// TwinCAT 3 PLC project ASRS_2
// ProgramVersion: 3.1.4024.0
// libraries:
//   Tc2_Standard, * (Beckhoff Automation GmbH)
//   Tc2_System, * (Beckhoff Automation GmbH)
//   Tc3_Module, * (Beckhoff Automation GmbH)
// project tree:
//   DUTs/Enum/ E_ConveyorMode.TcDUT, E_DiverterState.TcDUT (not stored), E_CraneState.TcDUT (not stored), E_AisleMode.TcDUT (not stored), E_SlotStatus.TcDUT (not stored), E_WarehouseState.TcDUT (not stored)
//   DUTs/Structure/ ST_Parcel.TcDUT (not stored), ST_StorageSlot.TcDUT (not stored), ST_Position.TcDUT (not stored), ST_CraneJob.TcDUT (not stored), ST_HMI_Search.TcDUT
//   GVLs/ GVL_IO.TcGVL, GVL_Config.TcGVL (not stored), GVL_Warehouse.TcGVL
//   / PlcTask.TcTTO (not stored)
//   POUs/ Class Diagram.TcCD (not stored), FB_WareHouseController.TcPOU, MAIN.TcPOU
//   POUs/ITFs/ I_Conveyor.TcIO, I_Diverter.TcIO (not stored), I_Crane.TcIO (not stored)
//   POUs/Entity/ FB_Conveyor.TcPOU, FB_BiDirectionConveyor.TcPOU (not stored), FB_RAT.TcPOU, FB_Crane.TcPOU (not stored)
//   POUs/Controller/ FB_InFeedController.TcPOU, FB_LoopController.TcPOU, FB_AisleController.TcPOU (not stored), FB_CraneController.TcPOU (not stored), FB_OutFeedController.TcPOU
// (motion and I/O tree: see PLC project asrs_test)
// real-time tasks:
//   TASK PlcTask: cycle T#10ms, priority 20, ADS port 350
//   TASK PlcTask1: cycle T#10ms, priority 21, ADS port 351

// ---- DUTs/Enum/E_ConveyorMode.TcDUT
{attribute 'qualified_only'}
{attribute 'strict'}
TYPE E_ConveyorMode :
(
    IDLE              := 0,
    RUNNING_FORWARD   := 10,
    RUNNING_BACKWARD  := 20,
    FAULT             := 99
);
END_TYPE

// ---- DUTs/Structure/ST_HMI_Search.TcDUT
TYPE ST_HMI_Search :
STRUCT
    (* Input from Operator *)
    sSearchID       : STRING(20);   
    bTriggerSearch  : BOOL;         
    
    (* Output to HMI *)
    bMatchFound     : BOOL;         
    nFoundCol       : INT;          
    nFoundRow       : INT;          
    nFoundDepth     : INT;          
    
    (* Selection Detail for Popup *)
    stSelectedParcel : ST_Parcel;   
    eSelectedStatus  : E_SlotStatus;
END_STRUCT
END_TYPE

// ---- GVLs/GVL_IO.TcGVL
{attribute 'qualified_only'}
VAR_GLOBAL
    // Infeed conveyor
    bInfeedSensor           : BOOL;
    bInfeedBlocker          : BOOL;
    bInfeedMotor            : BOOL;

    // Infeed RAT (transfers parcel from infeed conveyor onto loop)
    bInfeedRatSensor        : BOOL;
    bInfeedRatLift          : BOOL;
    bInfeedRatTravel        : BOOL;
    bInfeedRatUp            : BOOL;
    bInfeedRatDown          : BOOL;

    // Main loop conveyor
    bLoopMotor              : BOOL;
    bLoopSensor             : BOOL;

    // Aisle 1 junction on loop
    bAisle1ApproachSensor   : BOOL;
    bAisle1StopBlocker      : BOOL;
    bAisle1RatLift          : BOOL;
    bAisle1RatTravel        : BOOL;
    bRat1Sensor             : BOOL;
    bRat1Up                 : BOOL;
    bRat1Down               : BOOL;

    // Aisle 2 junction on loop
    bAisle2ApproachSensor   : BOOL;
    bAisle2StopBlocker      : BOOL;
    bAisle2RatLift          : BOOL;
    bAisle2RatTravel        : BOOL;
    bRat2Sensor             : BOOL;
    bRat2Up                 : BOOL;
    bRat2Down               : BOOL;

    // Outfeed junction on loop
    bOutfeedApproachSensor  : BOOL;
	bOutfeedExitSensor      : BOOL;
    bOutfeedStopBlocker     : BOOL;
    bOutfeedRatLift         : BOOL;
    bOutfeedRatTravel       : BOOL;
    bOutfeedRatSensor       : BOOL;
    bOutfeedRatUp           : BOOL;
    bOutfeedRatDown         : BOOL;

    // Aisle 1 conveyor
    bAisle1EntrySensor      : BOOL;
    bAisle1CraneStation     : BOOL;
    bAisle1MotorForward     : BOOL;
    bAisle1MotorReverse     : BOOL;

    // Aisle 2 conveyor
    bAisle2EntrySensor      : BOOL;
    bAisle2CraneStation     : BOOL;
    bAisle2MotorForward     : BOOL;
    bAisle2MotorReverse     : BOOL;

    // Outfeed conveyor
    bOutfeedSensor          : BOOL;
    bOutfeedMotor           : BOOL;

    // Crane 1
    fCrane1PosX             : LREAL;
    fCrane1PosY             : LREAL;
    bCrane1ForksExtended    : BOOL;
    bCrane1ForksHome        : BOOL;
    bCrane1MotorX           : BOOL;
    bCrane1MotorY           : BOOL;
    bCrane1ForksOut         : BOOL;
    bCrane1EStop            : BOOL;

    // Crane 2
    fCrane2PosX             : LREAL;
    fCrane2PosY             : LREAL;
    bCrane2ForksExtended    : BOOL;
    bCrane2ForksHome        : BOOL;
    bCrane2MotorX           : BOOL;
    bCrane2MotorY           : BOOL;
    bCrane2ForksOut         : BOOL;
    bCrane2EStop            : BOOL;
END_VAR

// ---- GVLs/GVL_Warehouse.TcGVL
{attribute 'qualified_only'}
VAR_GLOBAL PERSISTENT
    arrRack              : ARRAY[1..10, 1..4] OF ST_StorageSlot;
    nTotalStoredCount    : UDINT;
    nTotalRetrievedCount : UDINT;
    sWarehouseName       : STRING := 'IntimeTec_ASRS_01';
    bRackInitialized     : BOOL;
END_VAR

VAR_GLOBAL
    bSystemAutoMode      : BOOL := FALSE;
    bEmergencyStop       : BOOL := FALSE;
    sSystemStatusMsg     : STRING(80) := 'System Ready';
    stHmiSearch          : ST_HMI_Search;
END_VAR

// ---- POUs/ITFs/I_Conveyor.TcIO
INTERFACE I_Conveyor

PROPERTY bError : BOOL
GET
END_GET
END_PROPERTY

PROPERTY bMotorRun : BOOL
GET
END_GET
END_PROPERTY

PROPERTY bMotorReverse : BOOL
GET
END_GET
END_PROPERTY

METHOD M_Run
VAR_INPUT
    bForward : BOOL;
END_VAR
END_METHOD

METHOD M_Stop
VAR_INPUT
END_VAR
END_METHOD

METHOD M_Reset
VAR_INPUT
END_VAR
END_METHOD

END_INTERFACE

// ---- POUs/MAIN.TcPOU
PROGRAM MAIN
VAR
    fbWarehouse : FB_WareHouseController;
    bFirstScan  : BOOL := TRUE;
END_VAR

IF bFirstScan THEN
    GVL_Warehouse.bSystemAutoMode := FALSE;
    GVL_Warehouse.bEmergencyStop  := FALSE;
    GVL_Warehouse.sSystemStatusMsg:= 'System Ready';
    IF NOT GVL_Warehouse.bRackInitialized THEN
        fbWarehouse.M_InitRack();
    END_IF
    bFirstScan := FALSE;
END_IF

fbWarehouse();

END_PROGRAM

// ---- POUs/FB_WareHouseController.TcPOU
FUNCTION_BLOCK FB_WareHouseController
VAR_OUTPUT
    bError  : BOOL;
    eState  : E_WarehouseState := E_WarehouseState.IDLE;
END_VAR
VAR
    // ── Concrete entities (only instantiated here) ────────────────────────
    fbInfeedBelt    : FB_Conveyor;
    fbLoopBelt      : FB_Conveyor;
    fbAisle1Belt    : FB_BiDirectionConveyor;
    fbAisle2Belt    : FB_BiDirectionConveyor;
    fbOutfeedBelt   : FB_Conveyor;
    fbInfeedRat     : FB_RAT;
    fbAisle1Rat     : FB_RAT;
    fbAisle2Rat     : FB_RAT;
    fbOutfeedRat    : FB_RAT;
    fbCrane1        : FB_Crane;
    fbCrane2        : FB_Crane;

    // ── Controllers (receive interfaces via VAR_IN_OUT) ───────────────────
    fbInfeed        : FB_InFeedController;
    fbLoop          : FB_LoopController;
    fbAisle1        : FB_AisleController;
    fbAisle2        : FB_AisleController;
    fbCraneCtrl1    : FB_CraneController;
    fbCraneCtrl2    : FB_CraneController;
    fbOutfeed       : FB_OutFeedController;

    // ── Job queue ─────────────────────────────────────────────────────────
    arrJobs         : ARRAY[1..20] OF ST_CraneJob;
    nHead           : INT := 1;
    nTail           : INT := 1;
    nCount          : INT := 0;

    nTargetAisle    : INT := 0;
    bOutfeedReq     : BOOL;
END_VAR

// ── 1. Run all entities with their physical IO ────────────────────────────
fbInfeedBelt();
fbLoopBelt();

fbAisle1Belt(
    bEntrySensor        := GVL_IO.bAisle1EntrySensor,
    bCraneStationSensor := GVL_IO.bAisle1CraneStation
);
fbAisle2Belt(
    bEntrySensor        := GVL_IO.bAisle2EntrySensor,
    bCraneStationSensor := GVL_IO.bAisle2CraneStation
);
fbOutfeedBelt();

fbInfeedRat(
    bSensorOccupied := GVL_IO.bInfeedRatSensor,
    bSensorIsUp     := GVL_IO.bInfeedRatUp,
    bSensorIsDown   := GVL_IO.bInfeedRatDown
);
fbAisle1Rat(
    bSensorOccupied := GVL_IO.bRat1Sensor,
    bSensorIsUp     := GVL_IO.bRat1Up,
    bSensorIsDown   := GVL_IO.bRat1Down
);
fbAisle2Rat(
    bSensorOccupied := GVL_IO.bRat2Sensor,
    bSensorIsUp     := GVL_IO.bRat2Up,
    bSensorIsDown   := GVL_IO.bRat2Down
);
fbOutfeedRat(
    bSensorOccupied := GVL_IO.bOutfeedRatSensor,
    bSensorIsUp     := GVL_IO.bOutfeedRatUp,
    bSensorIsDown   := GVL_IO.bOutfeedRatDown
);

fbCrane1(
    fPosX          := GVL_IO.fCrane1PosX,
    fPosY          := GVL_IO.fCrane1PosY,
    bForksHome     := GVL_IO.bCrane1ForksHome,
    bForksExtended := GVL_IO.bCrane1ForksExtended
);
fbCrane2(
    fPosX          := GVL_IO.fCrane2PosX,
    fPosY          := GVL_IO.fCrane2PosY,
    bForksHome     := GVL_IO.bCrane2ForksHome,
    bForksExtended := GVL_IO.bCrane2ForksExtended
);

// ── 2. Write crane physical outputs ──────────────────────────────────────────
GVL_IO.bCrane1MotorX  := fbCrane1.bMotorX;
GVL_IO.bCrane1MotorY  := fbCrane1.bMotorY;
GVL_IO.bCrane1ForksOut:= fbCrane1.bForksOut;
GVL_IO.bCrane2MotorX  := fbCrane2.bMotorX;
GVL_IO.bCrane2MotorY  := fbCrane2.bMotorY;
GVL_IO.bCrane2ForksOut:= fbCrane2.bForksOut;

// ── 3. Emergency stop ─────────────────────────────────────────────────────────
IF GVL_Warehouse.bEmergencyStop THEN
    eState := E_WarehouseState.FAULT;
END_IF

IF eState = E_WarehouseState.FAULT THEN
    bError := TRUE;
    RETURN;
END_IF

// ── 4. Run controllers (dependency injection via VAR_IN_OUT) ─────────────────
fbInfeed(iInfeedBelt := fbInfeedBelt, iInfeedRat := fbInfeedRat);

fbLoop(
    nTargetAisle    := nTargetAisle,
    bOutfeedRequest := bOutfeedReq,
    iLoopBelt       := fbLoopBelt,
    iAisle1Rat      := fbAisle1Rat,
    iAisle2Rat      := fbAisle2Rat,
    iOutfeedRat     := fbOutfeedRat
);

fbAisle1(
    nAisleNumber    := 1,
    bInboundRequest := (nTargetAisle = 1) AND fbLoop.bLoopReady = FALSE,
    bOutboundRequest:= FALSE,
    bCranePickDone  := fbCraneCtrl1.bPickDone,
    bCraneDropDone  := fbCraneCtrl1.bDropDone,
    iAisleBelt      := fbAisle1Belt
);

fbAisle2(
    nAisleNumber    := 2,
    bInboundRequest := (nTargetAisle = 2) AND fbLoop.bLoopReady = FALSE,
    bOutboundRequest:= FALSE,
    bCranePickDone  := fbCraneCtrl2.bPickDone,
    bCraneDropDone  := fbCraneCtrl2.bDropDone,
    iAisleBelt      := fbAisle2Belt
);

fbCraneCtrl1(nAisleNumber := 1, iCrane := fbCrane1);
fbCraneCtrl2(nAisleNumber := 2, iCrane := fbCrane2);

fbOutfeed(iOutfeedBelt := fbOutfeedBelt);

// ── 5. Route incoming parcel ──────────────────────────────────────────────────
IF fbInfeed.bParcelReady THEN
    M_RouteParcel();
END_IF

// ── 6. Dispatch queued jobs to cranes ─────────────────────────────────────────
M_DispatchJobs();

// ── 7. HMI search ─────────────────────────────────────────────────────────────
IF GVL_Warehouse.stHmiSearch.bTriggerSearch THEN
    M_HmiSearch();
END_IF

// ── 8. Propagate errors ───────────────────────────────────────────────────────
bError := fbInfeed.bError OR fbLoop.bError OR fbAisle1.bError OR fbAisle2.bError
          OR fbCraneCtrl1.bError OR fbCraneCtrl2.bError OR fbOutfeed.bError;
IF bError THEN
    eState := E_WarehouseState.FAULT;
END_IF

METHOD PRIVATE M_DispatchJobs
VAR
    stJob : ST_CraneJob;
END_VAR
IF nCount = 0 THEN RETURN; END_IF

stJob := arrJobs[nHead];

IF stJob.nAisle = 1 AND NOT fbCraneCtrl1.bBusy THEN
    IF fbCraneCtrl1.M_AssignStore(stPos := stJob.stRackPos) THEN
        GVL_Warehouse.arrRack[stJob.stRackPos.nCol, stJob.stRackPos.nRow].eStatus := E_SlotStatus.OCCUPIED;
        arrJobs[nHead].bValid := FALSE;
        nHead  := nHead MOD 20 + 1;
        nCount := nCount - 1;
    END_IF
ELSIF stJob.nAisle = 2 AND NOT fbCraneCtrl2.bBusy THEN
    IF fbCraneCtrl2.M_AssignStore(stPos := stJob.stRackPos) THEN
        GVL_Warehouse.arrRack[stJob.stRackPos.nCol, stJob.stRackPos.nRow].eStatus := E_SlotStatus.OCCUPIED;
        arrJobs[nHead].bValid := FALSE;
        nHead  := nHead MOD 20 + 1;
        nCount := nCount - 1;
    END_IF
END_IF
END_METHOD

METHOD PRIVATE M_Enqueue
VAR_INPUT
    stJob : ST_CraneJob;
END_VAR
IF nCount >= 20 THEN RETURN; END_IF
arrJobs[nTail] := stJob;
nTail  := nTail MOD 20 + 1;
nCount := nCount + 1;
END_METHOD

METHOD PRIVATE M_HmiSearch
VAR
    nCol : INT;
    nRow : INT;
END_VAR
GVL_Warehouse.stHmiSearch.bMatchFound := FALSE;
FOR nCol := 1 TO GVL_Config.MAX_COLUMNS DO
    FOR nRow := 1 TO GVL_Config.MAX_ROWS DO
        IF GVL_Warehouse.arrRack[nCol, nRow].eStatus = E_SlotStatus.OCCUPIED AND
           GVL_Warehouse.arrRack[nCol, nRow].stParcel.sID = GVL_Warehouse.stHmiSearch.sSearchID THEN
            GVL_Warehouse.stHmiSearch.bMatchFound      := TRUE;
            GVL_Warehouse.stHmiSearch.nFoundCol        := nCol;
            GVL_Warehouse.stHmiSearch.nFoundRow        := nRow;
            GVL_Warehouse.stHmiSearch.stSelectedParcel := GVL_Warehouse.arrRack[nCol, nRow].stParcel;
            GVL_Warehouse.stHmiSearch.eSelectedStatus  := GVL_Warehouse.arrRack[nCol, nRow].eStatus;
        END_IF
    END_FOR
END_FOR
GVL_Warehouse.stHmiSearch.bTriggerSearch := FALSE;
END_METHOD

METHOD M_InitRack
VAR
    nCol : INT;
    nRow : INT;
END_VAR
FOR nCol := 1 TO GVL_Config.MAX_COLUMNS DO
    FOR nRow := 1 TO GVL_Config.MAX_ROWS DO
        GVL_Warehouse.arrRack[nCol, nRow].eStatus     := E_SlotStatus.EMPTY;
        GVL_Warehouse.arrRack[nCol, nRow].bMaintenance:= FALSE;
        // Even rows are rear/deep slots
        GVL_Warehouse.arrRack[nCol, nRow].bIsRear     := (nRow MOD 2 = 0);
    END_FOR
END_FOR
GVL_Warehouse.bRackInitialized := TRUE;
END_METHOD

METHOD M_RequestRetrieval : BOOL
VAR_INPUT
    nCol : INT;
    nRow : INT;
END_VAR
VAR
    stJob : ST_CraneJob;
END_VAR
IF nCol < 1 OR nCol > GVL_Config.MAX_COLUMNS OR
   nRow < 1 OR nRow > GVL_Config.MAX_ROWS THEN
    M_RequestRetrieval := FALSE;
    RETURN;
END_IF

IF GVL_Warehouse.arrRack[nCol, nRow].eStatus <> E_SlotStatus.OCCUPIED THEN
    M_RequestRetrieval := FALSE;
    RETURN;
END_IF

GVL_Warehouse.arrRack[nCol, nRow].eStatus := E_SlotStatus.RESERVED_OUT;

stJob.bValid             := TRUE;
stJob.bIsStore           := FALSE;
stJob.stParcel           := GVL_Warehouse.arrRack[nCol, nRow].stParcel;
stJob.stRackPos.nCol     := nCol;
stJob.stRackPos.nRow     := nRow;
stJob.stRackPos.fTargetX := (nCol - 1) * GVL_Config.COLUMN_SPACING;
stJob.stRackPos.fTargetY := (nRow - 1) * GVL_Config.ROW_SPACING;
stJob.nAisle             := SEL(stJob.stParcel.bIsHeavy, GVL_Config.CRANE1_AISLE, GVL_Config.CRANE2_AISLE);

M_Enqueue(stJob);
GVL_Warehouse.nTotalRetrievedCount := GVL_Warehouse.nTotalRetrievedCount + 1;
M_RequestRetrieval := TRUE;
END_METHOD

METHOD PRIVATE M_RouteParcel
VAR
    stJob  : ST_CraneJob;
    nCol   : INT;
    nRow   : INT;
    bFound : BOOL;
END_VAR
// Determine aisle by weight
IF fbInfeed.stParcel.bIsHeavy THEN
    nTargetAisle := GVL_Config.CRANE2_AISLE;
ELSE
    nTargetAisle := GVL_Config.CRANE1_AISLE;
END_IF

// Fill rear slots first (row 2, 4), then front (row 1, 3)
// Rear: row 2 and 4 (even rows = deep)
// Front: row 1 and 3 (odd rows = front)
bFound := FALSE;

// Pass 1: rear slots
FOR nCol := 1 TO GVL_Config.MAX_COLUMNS DO
    FOR nRow := 1 TO GVL_Config.MAX_ROWS DO
        IF GVL_Warehouse.arrRack[nCol, nRow].bIsRear
            AND GVL_Warehouse.arrRack[nCol, nRow].eStatus = E_SlotStatus.EMPTY
            AND NOT GVL_Warehouse.arrRack[nCol, nRow].bMaintenance THEN
            bFound := TRUE;
            EXIT;
        END_IF
    END_FOR
    IF bFound THEN EXIT; END_IF
END_FOR

// Pass 2: front slots if no rear slot found
IF NOT bFound THEN
    FOR nCol := 1 TO GVL_Config.MAX_COLUMNS DO
        FOR nRow := 1 TO GVL_Config.MAX_ROWS DO
            IF NOT GVL_Warehouse.arrRack[nCol, nRow].bIsRear
                AND GVL_Warehouse.arrRack[nCol, nRow].eStatus = E_SlotStatus.EMPTY
                AND NOT GVL_Warehouse.arrRack[nCol, nRow].bMaintenance THEN
                bFound := TRUE;
                EXIT;
            END_IF
        END_FOR
        IF bFound THEN EXIT; END_IF
    END_FOR
END_IF

IF NOT bFound THEN
    GVL_Warehouse.sSystemStatusMsg := 'Rack full';
    RETURN;
END_IF

GVL_Warehouse.arrRack[nCol, nRow].eStatus  := E_SlotStatus.RESERVED_IN;
GVL_Warehouse.arrRack[nCol, nRow].stParcel := fbInfeed.stParcel;

stJob.bValid             := TRUE;
stJob.bIsStore           := TRUE;
stJob.nAisle             := nTargetAisle;
stJob.stParcel           := fbInfeed.stParcel;
stJob.stRackPos.nCol     := nCol;
stJob.stRackPos.nRow     := nRow;
stJob.stRackPos.fTargetX := (nCol - 1) * GVL_Config.COLUMN_SPACING;
stJob.stRackPos.fTargetY := (nRow - 1) * GVL_Config.ROW_SPACING;

M_Enqueue(stJob);
GVL_Warehouse.nTotalStoredCount := GVL_Warehouse.nTotalStoredCount + 1;
GVL_Warehouse.sSystemStatusMsg  := 'Parcel stored';
END_METHOD

END_FUNCTION_BLOCK

// ---- POUs/Entity/FB_Conveyor.TcPOU
FUNCTION_BLOCK FB_Conveyor IMPLEMENTS I_Conveyor
VAR_OUTPUT
    bConveyorError        : BOOL;
    bConveyorMotorRun     : BOOL;
    bConveyorMotorReverse : BOOL;
END_VAR
VAR
    eMode       : E_ConveyorMode := E_ConveyorMode.IDLE;
    fbJamTimer  : TON;
END_VAR

//fbJamTimer(IN := bConveyorMotorRun, PT := GVL_Config.T_JAM_TIMEOUT);
IF fbJamTimer.Q THEN
    eMode := E_ConveyorMode.FAULT;
END_IF

CASE eMode OF
    E_ConveyorMode.IDLE:
        bConveyorMotorRun     := FALSE;
        bConveyorMotorReverse := FALSE;

    E_ConveyorMode.RUNNING_FORWARD:
        bConveyorMotorRun     := TRUE;
        bConveyorMotorReverse := FALSE;

    E_ConveyorMode.RUNNING_BACKWARD:
        bConveyorMotorRun     := TRUE;
        bConveyorMotorReverse := TRUE;

    E_ConveyorMode.FAULT:
        bConveyorMotorRun     := FALSE;
        bConveyorMotorReverse := FALSE;
        bConveyorError        := TRUE;
END_CASE

PROPERTY bError : BOOL
GET
bError := bConveyorError;
END_GET
END_PROPERTY

PROPERTY bMotorReverse : BOOL
GET
bMotorReverse := bConveyorMotorReverse;
END_GET
END_PROPERTY

PROPERTY bMotorRun : BOOL
GET
bMotorRun := bConveyorMotorRun;
END_GET
END_PROPERTY

METHOD M_Reset
VAR_INPUT
END_VAR
bConveyorError := FALSE;
eMode  := E_ConveyorMode.IDLE;
END_METHOD

METHOD M_Run
VAR_INPUT
    bForward : BOOL;
END_VAR
IF eMode = E_ConveyorMode.FAULT THEN RETURN; END_IF
IF bForward THEN
    eMode := E_ConveyorMode.RUNNING_FORWARD;
ELSE
    eMode := E_ConveyorMode.RUNNING_BACKWARD;
END_IF
END_METHOD

METHOD M_Stop
VAR_INPUT
END_VAR
eMode := E_ConveyorMode.IDLE;
END_METHOD

END_FUNCTION_BLOCK

// ---- POUs/Entity/FB_RAT.TcPOU
FUNCTION_BLOCK FB_RAT IMPLEMENTS I_Diverter
VAR_INPUT
    bSensorOccupied : BOOL;
    bSensorIsUp     : BOOL;
    bSensorIsDown   : BOOL;
END_VAR
VAR_OUTPUT
    bRatError          : BOOL;
    bIsLiftUp         : BOOL;
    bDivertMotorRun : BOOL;
END_VAR
VAR
    eRatState          : E_DiverterState := E_DiverterState.IDLE;
    fbLiftTimer     : TON;
    fbTravelTimer   : TON;
END_VAR

//fbLiftTimer(
//    IN := (eRatState = E_DiverterState.LIFTING OR eRatState = E_DiverterState.LOWERING),
//    PT := GVL_Config.T_RAT_LIFT_TIMEOUT
//);
//fbTravelTimer(IN := eRatState = E_DiverterState.DIVERTING, PT := T#6S);

IF fbLiftTimer.Q OR fbTravelTimer.Q THEN
    eRatState := E_DiverterState.FAULT;
END_IF

CASE eRatState OF
    E_DiverterState.IDLE:
        bIsLiftUp         := FALSE;
        bDivertMotorRun := FALSE;

    E_DiverterState.LIFTING:
        bIsLiftUp := TRUE;
        IF bSensorIsUp THEN
            eRatState := E_DiverterState.DIVERTING;
        END_IF

    E_DiverterState.DIVERTING:
        bIsLiftUp         := TRUE;
        bDivertMotorRun := TRUE;
        IF NOT bSensorOccupied THEN
            eRatState := E_DiverterState.LOWERING;
        END_IF

    E_DiverterState.LOWERING:
        bIsLiftUp         := FALSE;
        bDivertMotorRun := FALSE;
        IF bSensorIsDown THEN
            eRatState := E_DiverterState.DONE;
        END_IF
	
    E_DiverterState.FAULT:
        bIsLiftUp         := FALSE;
        bDivertMotorRun := FALSE;
        bRatError          := TRUE;
END_CASE

PROPERTY bError : BOOL
GET
bError := bRatError;
END_GET
END_PROPERTY

PROPERTY bLiftUp : BOOL
GET
bLiftUp := bIsLiftUp;
END_GET
END_PROPERTY

PROPERTY bTravelMotorRun : BOOL
GET
bTravelMotorRun := bDivertMotorRun;
END_GET
END_PROPERTY

PROPERTY eState : E_DiverterState
GET
eState := eRatState;
END_GET
END_PROPERTY

METHOD M_Divert
VAR_INPUT
END_VAR
IF eRatState = E_DiverterState.IDLE THEN
    eRatState := E_DiverterState.LIFTING;
END_IF
END_METHOD

METHOD M_Stop
VAR_INPUT
END_VAR
bIsLiftUp         := FALSE;
bDivertMotorRun := FALSE;
eRatState          := E_DiverterState.IDLE;
END_METHOD

END_FUNCTION_BLOCK

// ---- POUs/Controller/FB_InFeedController.TcPOU
FUNCTION_BLOCK FB_InFeedController
VAR_OUTPUT
    bParcelReady    : BOOL;
    bError          : BOOL;
    stParcel        : ST_Parcel;
	
END_VAR
VAR_INPUT
	iInfeedBelt     : I_Conveyor;
    iInfeedRat      : I_Diverter;
END_VAR
VAR
    nState : (IDLE, CONVEYING, WAIT_RAT_CLEAR, DONE) := IDLE;
END_VAR

// Write physical outputs
GVL_IO.bInfeedMotor   := iInfeedBelt.bMotorRun;
GVL_IO.bInfeedRatLift := iInfeedRat.bLiftUp;
GVL_IO.bInfeedRatTravel := iInfeedRat.bTravelMotorRun;

CASE nState OF

    IDLE:
        bParcelReady := FALSE;
        // Parcel arrived at infeed sensor
        IF GVL_IO.bInfeedSensor THEN
            // Stop parcel with blocker if infeed RAT is busy
            GVL_IO.bInfeedBlocker := iInfeedRat.eState = E_DiverterState.IDLE;
            IF GVL_IO.bInfeedBlocker THEN
                iInfeedBelt.M_Run(bForward := TRUE);
                nState := CONVEYING;
				GVL_IO.bInfeedBlocker := FALSE;
            END_IF
        END_IF

    CONVEYING:
        // Belt running, move parcel toward RAT
        // When parcel reaches RAT position, stop belt and divert
        IF GVL_IO.bInfeedRatSensor THEN
            iInfeedBelt.M_Stop();
            iInfeedRat.M_Divert();
            nState := WAIT_RAT_CLEAR;
        END_IF

    WAIT_RAT_CLEAR:
        // Wait for RAT to complete divert and return to idle
        IF NOT GVL_IO.bInfeedRatSensor THEN
            bParcelReady := TRUE;
			GVL_IO.bInfeedRatSensor := FALSE;
            nState := DONE;
        END_IF

    DONE:
        // Warehouse controller reads stParcel and clears bParcelReady
        IF NOT bParcelReady THEN
            nState := IDLE;
        END_IF

END_CASE

bError := iInfeedRat.bError OR iInfeedBelt.bError;

END_FUNCTION_BLOCK

// ---- POUs/Controller/FB_LoopController.TcPOU
FUNCTION_BLOCK FB_LoopController
VAR_INPUT
    nTargetAisle    : INT;
    bOutfeedRequest : BOOL;
	iLoopBelt       : I_Conveyor;
    iAisle1Rat      : I_Diverter;
    iAisle2Rat      : I_Diverter;
    iOutfeedRat     : I_Diverter;
END_VAR
VAR_OUTPUT
    bLoopReady      : BOOL;
    bError          : BOOL;
END_VAR

VAR
    nState : (MONITORING, DIVERT_A1, DIVERT_A2, DIVERT_OUT) := MONITORING;
END_VAR

// Write physical outputs
GVL_IO.bLoopMotor          := iLoopBelt.bMotorRun;
GVL_IO.bAisle1RatLift      := iAisle1Rat.bLiftUp;
GVL_IO.bAisle1RatTravel    := iAisle1Rat.bTravelMotorRun;
GVL_IO.bAisle2RatLift      := iAisle2Rat.bLiftUp;
GVL_IO.bAisle2RatTravel    := iAisle2Rat.bTravelMotorRun;
GVL_IO.bOutfeedRatLift     := iOutfeedRat.bLiftUp;
GVL_IO.bOutfeedRatTravel   := iOutfeedRat.bTravelMotorRun;

CASE nState OF

    MONITORING:
        bLoopReady := TRUE;
        iLoopBelt.M_Run(bForward := TRUE);

        // Parcel at Aisle 1 junction and Aisle 1 is the target
        IF GVL_IO.bAisle1ApproachSensor AND nTargetAisle = 1
            AND iAisle1Rat.eState = E_DiverterState.IDLE THEN
            GVL_IO.bAisle1StopBlocker := TRUE;
            nState := DIVERT_A1;

        // Parcel at Aisle 2 junction and Aisle 2 is the target
        ELSIF GVL_IO.bAisle2ApproachSensor AND nTargetAisle = 2
            AND iAisle2Rat.eState = E_DiverterState.IDLE THEN
            GVL_IO.bAisle2StopBlocker := TRUE;
            nState := DIVERT_A2;

        // Parcel at outfeed junction
        ELSIF GVL_IO.bOutfeedApproachSensor AND bOutfeedRequest
            AND iOutfeedRat.eState = E_DiverterState.IDLE THEN
            GVL_IO.bOutfeedStopBlocker := TRUE;
            nState := DIVERT_OUT;
        END_IF

    DIVERT_A1:
        bLoopReady := FALSE;
        // Parcel centered on RAT sensor - execute divert
        IF GVL_IO.bRat1Sensor THEN
            iLoopBelt.M_Stop();
            GVL_IO.bAisle1StopBlocker := FALSE;
            iAisle1Rat.M_Divert();
        END_IF
        IF iAisle1Rat.eState = E_DiverterState.DONE AND NOT GVL_IO.bRat1Sensor THEN
			iAisle1Rat.M_Stop();
            nState := MONITORING;
        END_IF

    DIVERT_A2:
        bLoopReady := FALSE;
        IF GVL_IO.bRat2Sensor THEN
            iLoopBelt.M_Stop();
            GVL_IO.bAisle2StopBlocker := FALSE;
            iAisle2Rat.M_Divert();
        END_IF
        IF iAisle2Rat.eState = E_DiverterState.DONE AND NOT GVL_IO.bRat2Sensor THEN
			iAisle2Rat.M_Stop();
            nState := MONITORING;
        END_IF

    DIVERT_OUT:
        bLoopReady := FALSE;
        IF GVL_IO.bOutfeedRatSensor THEN
            iLoopBelt.M_Stop();
            GVL_IO.bOutfeedStopBlocker := FALSE;
            iOutfeedRat.M_Divert();
        END_IF
        IF iOutfeedRat.eState = E_DiverterState.IDLE AND NOT GVL_IO.bOutfeedRatSensor THEN
            nState := MONITORING;
        END_IF

END_CASE

bError := iLoopBelt.bError OR iAisle1Rat.bError OR iAisle2Rat.bError OR iOutfeedRat.bError;

END_FUNCTION_BLOCK

// ---- POUs/Controller/FB_OutFeedController.TcPOU
FUNCTION_BLOCK FB_OutFeedController
VAR_OUTPUT
    bBusy           : BOOL;
    bError          : BOOL;
    bComplete       : BOOL;
	
END_VAR
VAR
    nState : (IDLE, RUNNING, DONE) := IDLE;
END_VAR
VAR_INPUT
	iOutfeedBelt    : I_Conveyor;
END_VAR

GVL_IO.bOutfeedMotor := iOutfeedBelt.bMotorRun;

CASE nState OF

    IDLE:
        bBusy     := FALSE;
        bComplete := FALSE;
        // Parcel appears at outfeed sensor after loop RAT diverted it
        IF GVL_IO.bOutfeedApproachSensor AND NOT GVL_IO.bOutfeedExitSensor THEN
            iOutfeedBelt.M_Run(bForward := TRUE);
            bBusy  := TRUE;
            nState := RUNNING;
        END_IF

    RUNNING:
        // Run until parcel clears the exit sensor
        IF GVL_IO.bOutfeedExitSensor THEN
            iOutfeedBelt.M_Stop();
            bComplete := TRUE;
            nState    := DONE;
        END_IF

    DONE:
        bBusy  := FALSE;
        nState := IDLE;

END_CASE

bError := iOutfeedBelt.bError;

END_FUNCTION_BLOCK
